FUNCTION_BLOCK QueryService (* Query Service Function Block *)
  (* Standard: 61499-2; Description: Copyright (c) 2018 fortiss GmbH This program and the accompanying materials are made available under the terms of the Eclipse Public License 2.0 which is available at https://www.eclipse.org/legal/epl-2.0/ SPDX-License-Identifier: EPL-2.0 *)
  (* Version 1.0, 2018-09-21, Jose Cabral, fortiss GmbH *)
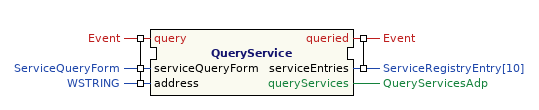
  EVENT_INPUT
    query WITH serviceQueryForm, address; (* Query for services *)
  END_EVENT
  EVENT_OUTPUT
    queried WITH serviceEntries; (* Query finished *)
  END_EVENT
  VAR_INPUT
    serviceQueryForm : ServiceQueryForm; (* The Arrowhead Service object that is looked for (SD and supported IDD-s) *)
    address : WSTRING; (* Address of the Service Registry (not officially in the documentation, but it simplifies the FBs) *)
  END_VAR
  VAR_OUTPUT
    serviceEntries : ARRAY [0..9] OF ServiceRegistryEntry; (* Result of the query request *)
  END_VAR
  PLUGS
    queryServices : QueryServicesAdp; (* Query Services adapter *)
  END_PLUGS
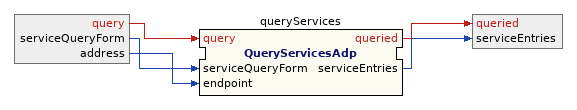
  EVENT_CONNECTIONS
    query TO queryServices.query;
    queryServices.queried TO queried;
  END_CONNECTIONS
  DATA_CONNECTIONS
    serviceQueryForm TO queryServices.serviceQueryForm;
    queryServices.serviceEntries TO serviceEntries;
    address TO queryServices.endpoint;
  END_CONNECTIONS
END_FUNCTION_BLOCK
